VAR_GLOBAL
	
{attribute 'pytmc' :=' pv: EM2K0:XGMD:OVERRIDE_INJ '}
	xOverrideMode : BOOL:= false;
	
	{attribute 'pytmc' :=' pv: EM2K0:XGMD:GHC:50 '}
	GHC_50 : FB_ITR90;	
	
	{attribute 'pytmc' :=' pv: EM2K0:XGMD:VCN:50 '}
	VCN_50 : FB_VCN;
	{attribute 'pytmc' :=' pv: EM2K0:XGMD:VGP:50 '}
	VGP_50 : FB_VGP;

	{attribute 'pytmc' :=' pv: EM2K0:XGMD:GCM:80 '}
	GCM_80 : FB_GCM;

	{attribute 'pytmc' :=' pv: EM2K0:XGMD:VVC:80 '}
	VVC_80:FB_VVC;
	{attribute 'pytmc' :=' pv: EM2K0:XGMD:VVC:81 '}
	VVC_81:FB_VVC;
	{attribute 'pytmc' :=' pv: EM2K0:XGMD:VVC:82 '}
	VVC_82:FB_VVC;
	{attribute 'pytmc' :=' pv: EM2K0:XGMD:VVC:83 '}
	VVC_83 : FB_VVC;
	{attribute 'pytmc' :=' pv: EM2K0:XGMD:VVC:84 '}
	VVC_84 : FB_VVC;
	{attribute 'pytmc' :=' pv: EM2K0:XGMD:VVC:85 '}
	VVC_85 : FB_VVC;
	{attribute 'pytmc' :=' pv: EM2K0:XGMD:VVC:86 '}
	VVC_86 : FB_VVC;
    {attribute 'pytmc' :=' pv: EM2K0:XGMD:VVC:87 '}
    {attribute 'TcLinkTo' := 	'.q_xOPN_DO	:=	TIIB[ES2004_03_08]^Channel 4^Output'}
	VVC_87 : FB_VVC;
//VVC87 KOS-DRL-02
// ES2004_03_08, pin: 8= 24V, 7=RTN
	
	(* Pressure Control*)
	{attribute 'pytmc' := ' pv: EM2K0:XGMD:GCP:50 '}
	GCP: ST_VG;
	{attribute 'pytmc' :=' pv: EM2K0:XGMD:CNTRL:SP;
	field: HOPR 1000;
	field: LOPR 0;
	field: PREC 2;
	field: EGU "TORR";
	'}
	fSetpointValue :REAL; 
	{attribute 'pytmc' :=' pv:  EM2K0:XGMD:CNTRL:GO;
	 field: ZNAM STOP; 
	 field: ONAM START; 
	 io: io;	'}
	bGo: BOOL; 
 	{attribute 'pytmc' :=' pv: EM2K0:XGMD:CNTRL:RESET;
	 field: ZNAM FALSE; 
	 field: ONAM TRUE; 
	 io: io;
	 '}
	bReset : BOOL; 
	{attribute 'pytmc' :=' pv:  EM2K0:XGMD:CNTRL:ERROR;
    field: ZNAM FALSE; 
	 field: ONAM TRUE; 
	 io: io;
	 '}
	bError : BOOL; 
	{attribute 'pytmc' :=' pv:  EM2K0:XGMDCNTRL:Kp1 '}
	fKp1 : REAL:= 0.5; 
	{attribute 'pytmc' :=' pv:  EM2K0:XGMD:CNTRL:Tn1 '}
	fTn1 : REAL:= 0.5; 
	{attribute 'pytmc' :=' pv:  EM2K0:XGMD:CNTRL:Kp2 '}
	fKp2 : REAL:= 0.01; 
	{attribute 'pytmc' :=' pv:  EM2K0:XGMD:CNTRL:Tn2 '}
	fTn2 : REAL:= 0.5; 
	
	(*Additional VCN Interlock*)
	{attribute 'pytmc' :=' pv:  EM2K0:XGMD:VCN_ILK;
    field: ZNAM FALSE; 
	 field: ONAM TRUE; 
	 io: io;
	 '}
	bAdditionalVCNIlk : BOOL:=TRUE; 
	
	(*HV*)
	{attribute 'pytmc' :=' pv: EM2K0:XGMD:PSV:1 '}
	hv1 : FB_HighVoltage;
	//{attribute 'pytmc' :=' pv: EM2K0:XGMD:PSV '}	
	//hv2 : FB_HighVoltage;
	
	(*RTD*)
	
	{attribute 'pytmc' :=' pv: EM2K0:XGMD:RTD:1 '}
	{attribute 'TcLinkTo' := '.iRaw := TIIB[EL3202_03_08]^RTD Inputs Channel 1^Value;
                              .bError := TIIB[EL3202_03_08]^RTD Inputs Channel 1^Status^Error;
                              .bUnderrange := TIIB[EL3202_03_08]^RTD Inputs Channel 1^Status^Underrange;
                              .bOverrange := TIIB[EL3202_03_08]^RTD Inputs Channel 1^Status^Overrange'}
	RTD_1 : FB_TempSensor;
	
	{attribute 'pytmc' :=' pv: EM2K0:XGMD:RTD:2 '}
	{attribute 'TcLinkTo' := '.iRaw := TIIB[EL3202_03_08]^RTD Inputs Channel 2^Value;
                              .bError := TIIB[EL3202_03_08]^RTD Inputs Channel 2^Status^Error;
                              .bUnderrange := TIIB[EL3202_03_08]^RTD Inputs Channel 2^Status^Underrange;
                              .bOverrange := TIIB[EL3202_03_08]^RTD Inputs Channel 2^Status^Overrange'}
	RTD_2 : FB_TempSensor;
	
END_VAR

(* stored: Version 1.1.0.1, ProductVersion 3.1.4022.18
   GVL GVL_Devices: Id {49019085-0c45-46f1-a256-56d701fd306c} *)
